{attribute 'qualified_only'}
VAR_GLOBAL RETAIN
	
    {attribute 'pytmc' := '
        pv: @(BTPS):Config:MaxFrameTime
        field: DESC Maximum delay from frame to frame
        field: EGU sec
    '}
    fMaximumFrameTime : LREAL;

END_VAR

(* stored: Version 1.1.0.1, ProductVersion 3.1.4022.18
   GVL GVL_BTPS_Retain: Id {f0024ece-4974-431e-ba4d-97ca2c5cbb7d} *)
